FUNCTION_BLOCK Test_AssertEquals_LINT EXTENDS TUnitTestBase
VAR
    AssertionUnderTest : TAssertion(AssertionListenerMock);
    AssertionListenerMock : TAssertionListenerMock;
    LINT_Variable : LINT := 1111;
END_VAR

AssertionListenerMock.AssertionFailed  := FALSE;
AssertionListenerMock.AssertionMessage := '';
AssertionListenerMock.ExpectedAsString := '';
AssertionListenerMock.ActualAsString   := '';

// Test the assertion...
AssertionUnderTest.AssertEquals_LINT(
    Expected := 2222,
    Actual   := LINT_Variable,
    VariableName := 'LINT_Variable');
 
    
// Check the assertion worked...    
Assertion.AssertEquals_BOOL(
    Expected := TRUE,
    Actual   := AssertionListenerMock.AssertionFailed,
    VariableName := 'AssertionListenerMock.AssertionFailed');

// Check the assertion messages...    
Assertion.AssertEquals_STRING(
    Expected := 'AssertEquals_LINT failed in AssertionTest: Value "LINT_Variable"',
    Actual   := AssertionListenerMock.AssertionMessage,
    VariableName := 'AssertionListenerMock.AssertionMessage');

Assertion.AssertEquals_STRING(
    Expected := '  Expected = 2222',
    Actual   := AssertionListenerMock.ExpectedAsString,
    VariableName := 'AssertionListenerMock.ExpectedAsString');

Assertion.AssertEquals_STRING(
    Expected := '  Actual   = 1111',
    Actual   := AssertionListenerMock.ActualAsString,
    VariableName := 'AssertionListenerMock.ActualAsString');

TestFinished();

END_FUNCTION_BLOCK

(* stored: Version 1.1.0.1, ProductVersion 3.1.4024.4
   POU Test_AssertEquals_LINT: Id {f19b24fa-5cf2-47d0-825e-be6487454fa3}, SpecialFunc None *)
